INTERFACE I_PushButton

PROPERTY IsPressed : Bool
GET
END_GET
END_PROPERTY

PROPERTY IsReleased : Bool
GET
END_GET
END_PROPERTY

END_INTERFACE

(* stored: Version 1.1.0.1, ProductVersion 3.1.4024.11
   Itf I_PushButton: Id {88b6f8ce-b56a-4e38-adcf-c359f3863b3b}
   Property IsPressed: Id {38d739b5-114b-4a0b-805d-a9a58d4242f1}
   Get Get: Id {393716ad-3acd-450b-86d5-74813ff16d89}
   Property IsReleased: Id {0d54dc67-7eeb-48cd-b166-831ecf010556}
   Get Get: Id {1816071d-c8ab-457d-a227-73332f8a8edd} *)
